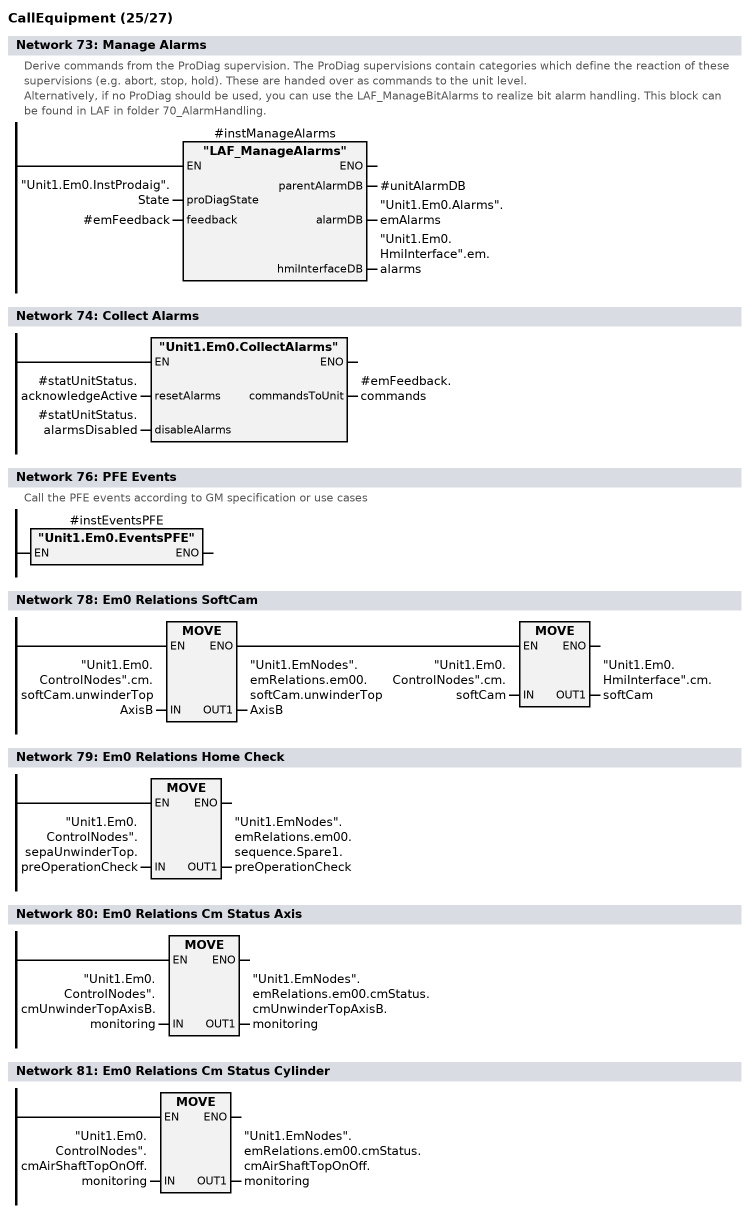
   RUNG wire#powerrail
      #instManageAlarms(proDiagState := "Unit1.Em0.InstProdaig".State, feedback := #emFeedback, parentAlarmDB => #unitAlarmDB, alarmDB => "Unit1.Em0.Alarms".emAlarms, hmiInterfaceDB => "Unit1.Em0.HmiInterface".em.alarms)
   END_RUNG
   // the same network as SCL:
   #instManageAlarms(proDiagState := "Unit1.Em0.InstProdaig".State,   // "LAF_ManageAlarms"
                     feedback := #emFeedback,
                     parentAlarmDB => #unitAlarmDB,
                     alarmDB => "Unit1.Em0.Alarms".emAlarms,
                     hmiInterfaceDB => "Unit1.Em0.HmiInterface".em.alarms);
END_REGION

REGION Network 74: Collect Alarms
   RUNG wire#powerrail
      "Unit1.Em0.CollectAlarms"(resetAlarms := #statUnitStatus.acknowledgeActive, disableAlarms := #statUnitStatus.alarmsDisabled, commandsToUnit => #emFeedback.commands)
   END_RUNG
   // the same network as SCL:
   "Unit1.Em0.CollectAlarms"(resetAlarms := #statUnitStatus.acknowledgeActive,
                           disableAlarms := #statUnitStatus.alarmsDisabled,
                           commandsToUnit => #emFeedback.commands);
END_REGION

REGION Network 75: *************** PFE Events**********************************
END_REGION

REGION Network 76: PFE Events
   // Call the PFE events according to GM specification or use cases
   RUNG wire#powerrail
      #instEventsPFE()
   END_RUNG
   // the same network as SCL:
   #instEventsPFE();   // "Unit1.Em0.EventsPFE"
END_REGION

REGION Network 77: ******************** Unit Output ********************
END_REGION

REGION Network 78: Em0 Relations SoftCam
   RUNG wire#powerrail
      Move(in := "Unit1.Em0.ControlNodes".cm.softCam.unwinderTopAxisB, out1 => "Unit1.EmNodes".emRelations.em00.softCam.unwinderTopAxisB)
      Move(in := "Unit1.Em0.ControlNodes".cm.softCam, out1 => "Unit1.Em0.HmiInterface".cm.softCam)
   END_RUNG
   // the same network as SCL:
   "Unit1.EmNodes".emRelations.em00.softCam.unwinderTopAxisB := "Unit1.Em0.ControlNodes".cm.softCam.unwinderTopAxisB;
   "Unit1.Em0.HmiInterface".cm.softCam := "Unit1.Em0.ControlNodes".cm.softCam;
END_REGION

REGION Network 79: Em0 Relations Home Check
   RUNG wire#powerrail
      Move(in := "Unit1.Em0.ControlNodes".sepaUnwinderTop.preOperationCheck, out1 => "Unit1.EmNodes".emRelations.em00.sequence.Spare1.preOperationCheck)
   END_RUNG
   // the same network as SCL:
   "Unit1.EmNodes".emRelations.em00.sequence.Spare1.preOperationCheck := "Unit1.Em0.ControlNodes".sepaUnwinderTop.preOperationCheck;
END_REGION

REGION Network 80: Em0 Relations Cm Status Axis
   RUNG wire#powerrail
      Move(in := "Unit1.Em0.ControlNodes".cmUnwinderTopAxisB.monitoring, out1 => "Unit1.EmNodes".emRelations.em00.cmStatus.cmUnwinderTopAxisB.monitoring)
   END_RUNG
   // the same network as SCL:
   "Unit1.EmNodes".emRelations.em00.cmStatus.cmUnwinderTopAxisB.monitoring := "Unit1.Em0.ControlNodes".cmUnwinderTopAxisB.monitoring;
END_REGION

REGION Network 81: Em0 Relations Cm Status Cylinder
   RUNG wire#powerrail
      Move(in := "Unit1.Em0.ControlNodes".cmAirShaftTopOnOff.monitoring, out1 => "Unit1.EmNodes".emRelations.em00.cmStatus.cmAirShaftTopOnOff.monitoring)
   END_RUNG
   // the same network as SCL:
   "Unit1.EmNodes".emRelations.em00.cmStatus.cmAirShaftTopOnOff.monitoring := "Unit1.Em0.ControlNodes".cmAirShaftTopOnOff.monitoring;
END_REGION

REGION Network 82: Em0 Relations CmStatus Digital Signal
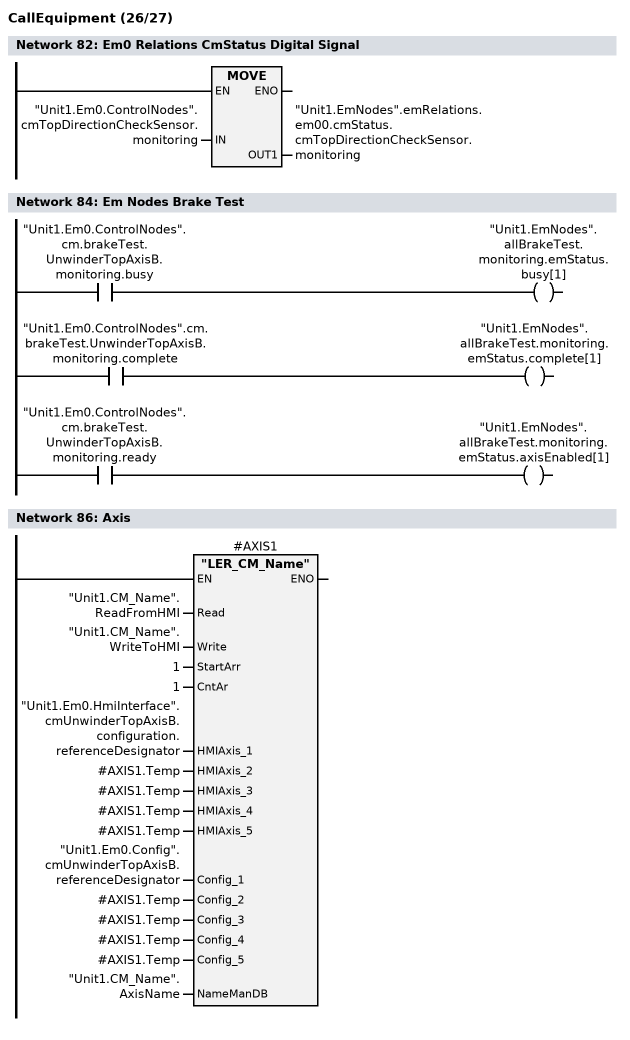
   RUNG wire#powerrail
      Move(in := "Unit1.Em0.ControlNodes".cmTopDirectionCheckSensor.monitoring, out1 => "Unit1.EmNodes".emRelations.em00.cmStatus.cmTopDirectionCheckSensor.monitoring)
   END_RUNG
   // the same network as SCL:
   "Unit1.EmNodes".emRelations.em00.cmStatus.cmTopDirectionCheckSensor.monitoring := "Unit1.Em0.ControlNodes".cmTopDirectionCheckSensor.monitoring;
END_REGION

REGION Network 83: Em0 Relations Sequence Interface
END_REGION

REGION Network 84: Em Nodes Brake Test
   RUNG wire#powerrail
      Contact( "Unit1.Em0.ControlNodes".cm.brakeTest.UnwinderTopAxisB.monitoring.busy )
      Coil( "Unit1.EmNodes".allBrakeTest.monitoring.emStatus.busy[1] )
   END_RUNG
   RUNG wire#powerrail
      Contact( "Unit1.Em0.ControlNodes".cm.brakeTest.UnwinderTopAxisB.monitoring.complete )
      Coil( "Unit1.EmNodes".allBrakeTest.monitoring.emStatus.complete[1] )
   END_RUNG
   RUNG wire#powerrail
      Contact( "Unit1.Em0.ControlNodes".cm.brakeTest.UnwinderTopAxisB.monitoring.ready )
      Coil( "Unit1.EmNodes".allBrakeTest.monitoring.emStatus.axisEnabled[1] )
   END_RUNG
   // the same network as SCL:
   "Unit1.EmNodes".allBrakeTest.monitoring.emStatus.busy[1] := "Unit1.Em0.ControlNodes".cm.brakeTest.UnwinderTopAxisB.monitoring.busy;
   "Unit1.EmNodes".allBrakeTest.monitoring.emStatus.complete[1] := "Unit1.Em0.ControlNodes".cm.brakeTest.UnwinderTopAxisB.monitoring.complete;
   "Unit1.EmNodes".allBrakeTest.monitoring.emStatus.axisEnabled[1] := "Unit1.Em0.ControlNodes".cm.brakeTest.UnwinderTopAxisB.monitoring.ready;
END_REGION

REGION Network 85 (SCL): SyncMotion Configuration
   REGION _name_
           "Unit1.MotionNodes".PLCToMotion.TechnologyObject.Axis.UnwinderTop := "Unit1.Em0.Config".axis[1];
           "Unit1.MotionNodes".PLCToMotion.Parameters.Dancer.Radius := "Unit1.Em0.ControlNodes".cmRadiusMeasure.monitoring.Radius;
           "Unit1.MotionNodes".PLCToMotion.Parameters.Dancer.UnwinderTopUse := "Unit1.EmNodes".emFeedback[0].isLinked;
   END_REGION
END_REGION

REGION Network 86: Axis
   RUNG wire#powerrail
      #AXIS1(Read := "Unit1.CM_Name".ReadFromHMI, Write := "Unit1.CM_Name".WriteToHMI, StartArr := 1, CntAr := 1, HMIAxis_1 := "Unit1.Em0.HmiInterface".cmUnwinderTopAxisB.configuration.referenceDesignator, HMIAxis_2 := #AXIS1.Temp, HMIAxis_3 := #AXIS1.Temp, HMIAxis_4 := #AXIS1.Temp, HMIAxis_5 := #AXIS1.Temp, Config_1 := "Unit1.Em0.Config".cmUnwinderTopAxisB.referenceDesignator, Config_2 := #AXIS1.Temp, Config_3 := #AXIS1.Temp, Config_4 := #AXIS1.Temp, Config_5 := #AXIS1.Temp, NameManDB := "Unit1.CM_Name".AxisName)
   END_RUNG
   // the same network as SCL:
   #AXIS1(Read := "Unit1.CM_Name".ReadFromHMI,   // "LER_CM_Name"
          Write := "Unit1.CM_Name".WriteToHMI,
          StartArr := 1,
          CntAr := 1,
          HMIAxis_1 := "Unit1.Em0.HmiInterface".cmUnwinderTopAxisB.configuration.referenceDesignator,
          HMIAxis_2 := #AXIS1.Temp,
          HMIAxis_3 := #AXIS1.Temp,
          HMIAxis_4 := #AXIS1.Temp,
          HMIAxis_5 := #AXIS1.Temp,
          Config_1 := "Unit1.Em0.Config".cmUnwinderTopAxisB.referenceDesignator,
          Config_2 := #AXIS1.Temp,
          Config_3 := #AXIS1.Temp,
          Config_4 := #AXIS1.Temp,
          Config_5 := #AXIS1.Temp,
          NameManDB := "Unit1.CM_Name".AxisName);
END_REGION

REGION Network 87: Cylinder
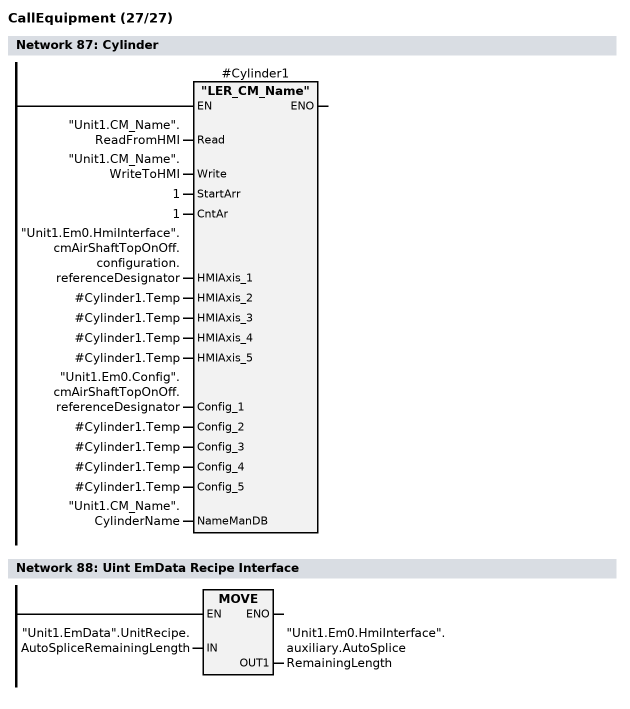
   RUNG wire#powerrail
      #Cylinder1(Read := "Unit1.CM_Name".ReadFromHMI, Write := "Unit1.CM_Name".WriteToHMI, StartArr := 1, CntAr := 1, HMIAxis_1 := "Unit1.Em0.HmiInterface".cmAirShaftTopOnOff.configuration.referenceDesignator, HMIAxis_2 := #Cylinder1.Temp, HMIAxis_3 := #Cylinder1.Temp, HMIAxis_4 := #Cylinder1.Temp, HMIAxis_5 := #Cylinder1.Temp, Config_1 := "Unit1.Em0.Config".cmAirShaftTopOnOff.referenceDesignator, Config_2 := #Cylinder1.Temp, Config_3 := #Cylinder1.Temp, Config_4 := #Cylinder1.Temp, Config_5 := #Cylinder1.Temp, NameManDB := "Unit1.CM_Name".CylinderName)
   END_RUNG
   // the same network as SCL:
   #Cylinder1(Read := "Unit1.CM_Name".ReadFromHMI,   // "LER_CM_Name"
              Write := "Unit1.CM_Name".WriteToHMI,
              StartArr := 1,
              CntAr := 1,
              HMIAxis_1 := "Unit1.Em0.HmiInterface".cmAirShaftTopOnOff.configuration.referenceDesignator,
              HMIAxis_2 := #Cylinder1.Temp,
              HMIAxis_3 := #Cylinder1.Temp,
              HMIAxis_4 := #Cylinder1.Temp,
              HMIAxis_5 := #Cylinder1.Temp,
              Config_1 := "Unit1.Em0.Config".cmAirShaftTopOnOff.referenceDesignator,
              Config_2 := #Cylinder1.Temp,
              Config_3 := #Cylinder1.Temp,
              Config_4 := #Cylinder1.Temp,
              Config_5 := #Cylinder1.Temp,
              NameManDB := "Unit1.CM_Name".CylinderName);
END_REGION

REGION Network 88: Uint EmData Recipe Interface
   RUNG wire#powerrail
      Move(in := "Unit1.EmData".UnitRecipe.AutoSpliceRemainingLength, out1 => "Unit1.Em0.HmiInterface".auxiliary.AutoSpliceRemainingLength)
   END_RUNG
   // the same network as SCL:
   "Unit1.Em0.HmiInterface".auxiliary.AutoSpliceRemainingLength := "Unit1.EmData".UnitRecipe.AutoSpliceRemainingLength;
END_REGION
END_FUNCTION_BLOCK
